// TwinCAT 3 PLC project PLC
// ProgramVersion: 3.1.4026.19
// CompilerDefines: VISU_USEPROPERTYINFO
// libraries:
//   Tc2_Standard, * (Beckhoff Automation GmbH)
//   Tc2_System, * (Beckhoff Automation GmbH)
// project tree:
//   / GlobalTextList.TcGTLO, PlcTask.TcTTO, Visualization Manager.TcVMO (not stored)
//   POUs/ FB_Motor.TcPOU, MAIN.TcPOU
//   VISUs/ Visualization.TcVIS
// real-time tasks:
//   TASK PlcTask: cycle T#10ms, priority 20, ADS port 350

CONFIGURATION PLC
    RESOURCE PLC ON TwinCAT3
        TASK PlcTask(INTERVAL := T#10ms, PRIORITY := 20);
        PROGRAM MAIN WITH PlcTask : MAIN;
    END_RESOURCE
END_CONFIGURATION

// ---- POUs/MAIN.TcPOU
PROGRAM MAIN
VAR
	fbBandMotor : FB_Motor;
	fbOfenMotor : FB_Motor;
	
	bBandStart : BOOL;
	bBandStop : BOOL;
	bBandErr : BOOL;
	bBandReset : BOOL;
	
	bOfenStart : BOOL;
	bOfenStop : BOOL;
	bOfenErr : BOOL;
	bOfenReset : BOOL;
END_VAR

fbBandMotor(
	bStart := bBandStart,
	bStop := bBandStop,
	bThermalErr := bBandErr,
	bReset := bBandReset
);

fbOfenMotor(
	bStart := bOfenStart,
	bStop := bOfenStop,
	bThermalErr := bOfenErr,
	bReset := bOfenReset
);

END_PROGRAM

// ---- POUs/FB_Motor.TcPOU
FUNCTION_BLOCK FB_Motor

VAR_INPUT
	bStart : BOOL;
	bStop : BOOL;
	bThermalErr : BOOL;
	bReset : BOOL;
END_VAR

VAR_OUTPUT
	bMotorRun : BOOL;
	bErrorLight : BOOL;
END_VAR

VAR
	
END_VAR

IF bThermalErr THEN
	bMotorRun := FALSE;
	bErrorLight := TRUE;
ELSIF bReset THEN
	bErrorLight := FALSE;
END_IF

IF NOT bErrorLight THEN
	
	IF bStop THEN
		bMotorRun := FALSE;
	ELSIF bStart THEN
		bMotorRun := TRUE;
	END_IF
	
ELSE
	bMotorRun := FALSE;
END_IF

END_FUNCTION_BLOCK

// ---- GlobalTextList.TcGTLO
TEXTLIST GlobalTextList
  174 = 'Band Information'
  36 = 'Error'
  974 = 'Error Light'
  252 = 'Ofen Information'
  682 = 'Reset'
  272 = 'Run'
  573 = 'Start'
  459 = 'Stop'
END_TEXTLIST

// ---- VISUs/Visualization.TcVIS
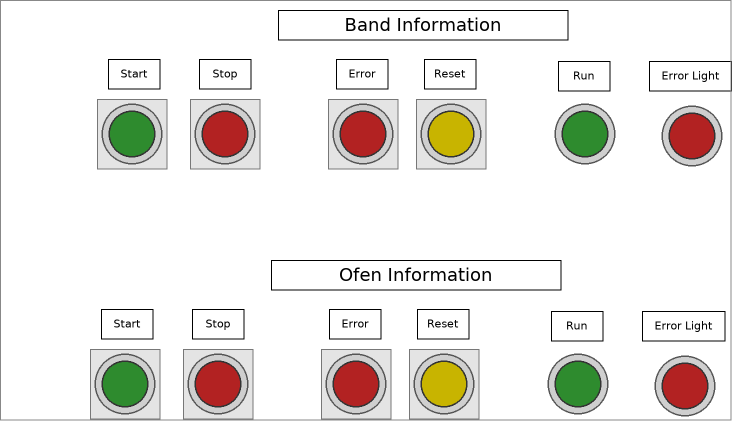
VISUALIZATION Visualization  // 732x421
    PushSwitch (97,99 70x70), variable: MAIN.bBandStart, behaviour: TOGGLE, style: Switch-PushSwitch-Green
    PushSwitch (190,99 70x70), variable: MAIN.bBandStop, behaviour: TOGGLE, style: Switch-PushSwitch-Red
    PushSwitch (328,99 70x70), variable: MAIN.bBandErr, behaviour: TOGGLE, style: Switch-PushSwitch-Red
    PushSwitch (416,99 70x70), variable: MAIN.bBandReset, behaviour: TOGGLE, style: Switch-PushSwitch-Yellow
    Lamp1 (550,99 70x70), variable: MAIN.fbBandMotor.bMotorRun, style: Lamp-Lamp1-Green
    Lamp1 (657,101 70x70), variable: MAIN.fbBandMotor.bErrorLight, style: Lamp-Lamp1-Red
    Rectangle (108,59 52x30), "Start"
    Rectangle (199,59 52x30), "Stop"
    Rectangle (336,59 52x30), "Error"
    Rectangle (424,59 52x30), "Reset"
    Rectangle (558,61 52x30), "Run"
    Rectangle (649,61 83x30), "Error Light"
    Rectangle (278,10 290x30), "Band Information"
    PushSwitch (90,349 70x70), variable: MAIN.bOfenStart, behaviour: TOGGLE, style: Switch-PushSwitch-Green
    PushSwitch (183,349 70x70), variable: MAIN.bOfenStop, behaviour: TOGGLE, style: Switch-PushSwitch-Red
    PushSwitch (321,349 70x70), variable: MAIN.bOfenErr, behaviour: TOGGLE, style: Switch-PushSwitch-Red
    PushSwitch (409,349 70x70), variable: MAIN.bOfenReset, behaviour: TOGGLE, style: Switch-PushSwitch-Yellow
    Lamp1 (543,349 70x70), variable: MAIN.fbOfenMotor.bMotorRun, style: Lamp-Lamp1-Green
    Lamp1 (650,351 70x70), variable: MAIN.fbOfenMotor.bErrorLight, style: Lamp-Lamp1-Red
    Rectangle (101,309 52x30), "Start"
    Rectangle (192,309 52x30), "Stop"
    Rectangle (329,309 52x30), "Error"
    Rectangle (417,309 52x30), "Reset"
    Rectangle (551,311 52x30), "Run"
    Rectangle (642,311 83x30), "Error Light"
    Rectangle (271,260 290x30), "Ofen Information"
END_VISUALIZATION
